# EPICS StreamDevice protocol: CM.proto
#####CRYOMECH protocol File
#SMDP SYCON

Terminator = CR;
ReplyTimeout = 1000;
locktimeout = 5000;
readtimeout  = 1000;
extrainput   = Ignore;

###################################################
#SET FUNCTIONS
###################################################
#        out "%B\xCA\xAA%B\x00\xAA%B\x01\xAA%B\x70\xAA%B\x00\xAA%B\x00\x8E";

#writes
StartComp{
   out "\x02\x10\x80\x61\xd5\x01\x00\x00\x00\x00\x01\x3c\x38";
}

StopComp{
   out "\x02\x10\x80\x61\xC5\x98\x00\x00\x00\x00\x01\x34\x3F";

}
###################################################
#READ FUNCTIONS
###################################################
ReadCompONOFF{
   out "\x02\x10\x80\x63\x5F\x95\x00\x3E\x37";
   in  "%*3r\x63\x5f\x95%*4r%r";
}

ReadINCoolantTemp {
   out "\x02\x10\x80\x63\x07\x31\x8F\x00\x38\x3F";
   in  "\x02\x10\x89\x63\x07\x31\x8F\x00%4r";
}

ReadOUTCoolantTemp {
   out "\x02\x10\x80\x63\x07\x31\x8F\x01\x39\x30";
   in  "\x02\x10\x89\x63\x07\x31\x8F\x01%4r";
}

ReadHeTemp{
   out "\x02\x10\x80\x63\x07\x31\x8F\x07\x30\x39\x31";
   in  "\x02\x10\x89\x63\x07\x31\x8F\x07\x30\x00%4r";
}

ReadOilTemp {
   out "\x02\x10\x80\x63\x07\x31\x8F\x03\x39\x32";
   in  "\x02\x10\x89\x63\x07\x31\x8F\x03%4r";
}

ReadHPressSide{
    out "\x02\x10\x80\x63\xAA\x50\x00\x3E\x3D";
    in  "\x02\x10\x89\x63\xAA\x50\x00%4r";
}

ReadLPressSide{
    out "\x02\x10\x80\x63\xAA\x50\x01\x3E\x3E";
    in  "\x02\x10\x89\x63\xAA\x50\x01%4r";
}

readCompressorID{
    out "\x02\x10\x80\x61\xD5\x01\x00\x00\x00\x00\x01\x3C\x38";
    in  "\x02\x10\x89\x63\xAA\x50\x01%4r";
}

ReadMotorCurrent{
    out "\x02\x10\x80\x63\x63\x8B\x00\x3E\x31";
    in  "\x02\x10\x89\x63\x63\x8B\x00%4r";
}

#0 no error else error or warning
ReadStatus{
    out "\x02\x10\x80\x63\x65\xA4\x00\x3F\x3C";
    in  "\x02\x10\x89\x63\x65\xA4\x00%4r";
}
